// TwinCAT 3 PLC project MqttTest
// Title: MqttTest
// Company: FactoryAutomation
// Author: Filippo Boido
// ProjectVersion: 1.4.2.8
// ProgramVersion: 3.1.4023.0
// libraries:
//   ChainControllerLib, * (FactoryAutomation)
//   MqttFramework, * (FactoryAutomation)
//   StateMachineLib, * (FactoryAutomation)
//   StepWorkerLib, * (FactoryAutomation)
//   Tc2_Standard, * (Beckhoff Automation GmbH)
//   Tc2_System, * (Beckhoff Automation GmbH)
//   Tc3_Module, * (Beckhoff Automation GmbH)
//   VisuSymbols,3.5.10.0,System
// project tree:
//   / GlobalTextList.TcGTLO (not stored), PlcTask.TcTTO, Version.TcPOU, Visualisierungsmanager.TcVMO (not stored)
//   POUs/Basic/Conveyors/ BeltConveyor.TcPOU, Conveyor.TcPOU, PalletizerConveyor.TcPOU, RollerConveyor.TcPOU
//   POUs/Basic/Cylinder/ Cylinder.TcPOU
//   POUs/Basic/Elevator/ Elevator.TcPOU, PalletizerElevator.TcPOU
//   POUs/Basic/Sensor/ Sensor.TcPOU
//   POUs/HeavyModules/LineRegulator/ SM_LineRegulator.TcPOU
//   POUs/HeavyModules/TransferLine/ TL_BUSY.TcDUT, TL_RollerConveyors.TcDUT (not stored), SM_TransferLine.TcPOU
//   POUs/HeavyModules/TransferLine/StepChains/BeltConveyors/ SC_ACTUATOR_BeltConveyors.TcDUT (not stored), SC_BUSY_BeltConveyors.TcDUT, SC_SENSOR_BeltConveyors.TcDUT (not stored), SC_BeltConveyors.TcPOU
//   POUs/HeavyModules/TransferLine/StepChains/PostPalletizer/ SC_PostPalletizer.TcPOU
//   POUs/HeavyModules/TransferLine/StepChains/PrePalletizer/ SC_PrePalletizer.TcPOU
//   POUs/LightModules/PresenceDetector/ PresenceDetector.TcPOU
//   POUs/LightModules/Turntable/ Turntable.TcPOU
//   POUs/Main/ MAIN_BUSY.TcDUT (not stored), MAIN.TcPOU
//   POUs/MediumModules/Palletizer/ PAL_Busy.TcDUT, SM_Palletizer.TcPOU
//   POUs/MediumModules/Palletizer/StepChains/FirstFloor/ SC_BUSY_FirstFloor.TcDUT (not stored), SC_FirstFloor.TcPOU
//   POUs/MediumModules/Palletizer/StepChains/SecondFloor/ SC_BUSY_SecondFloor.TcDUT, SC_SecondFloor.TcPOU
//   POUs/ Visu.TcPOU (not stored)
//   VISUs/ Visualization.TcVIS
// real-time tasks:
//   TASK PlcTask: cycle T#10ms, priority 20, ADS port 350

CONFIGURATION MqttTest
    RESOURCE PLC ON TwinCAT3
        TASK PlcTask(INTERVAL := T#10ms, PRIORITY := 20);
        PROGRAM MAIN WITH PlcTask : MAIN;
    END_RESOURCE
END_CONFIGURATION

// ---- POUs/HeavyModules/TransferLine/TL_BUSY.TcDUT

TYPE TL_BUSY :
(
	eTlBusyStart := 0,
	eTlStartEntranceConveyor,
	eTlStartUpwardsConveyor,
	eTlExecutePalletizer,
	eTlSignalError
)UINT;
END_TYPE

// ---- POUs/HeavyModules/TransferLine/StepChains/BeltConveyors/SC_BUSY_BeltConveyors.TcDUT

TYPE SC_BUSY_BeltConveyors :
(
	eBusySCStart := 0,
	eStartEntranceConveyor,
	eStartUpwardsConveyor,
	eExecutePalletizer,
	eStopEntranceConveyor,
	eWaitForPalletizer,
	eSignalError
)UINT;
END_TYPE

// ---- POUs/MediumModules/Palletizer/PAL_Busy.TcDUT

TYPE PAL_Busy :
(
	ePALStart := 0
	
	
);
END_TYPE

// ---- POUs/MediumModules/Palletizer/StepChains/SecondFloor/SC_BUSY_SecondFloor.TcDUT

TYPE SC_BUSY_SecondFloor :
(
	eSecondFloorStart := 0,
	eActivateTurn,
	eActivateBeltForw,
	eWaitForPackages,
	ePushPackages,
	eRetractPusher,
	eClamp,
	eRetractClamper,
	eWaitForPallet,
	eOpenPlate,
	eClosePlate,
	eElevatorUp,
	eElevatorDown,
	eStartChains,
	eStopChains,
	eWaitForFirstFloor,
	eSyncWithFirstFloor,
	eSecondFloorDone
);
END_TYPE

// ---- POUs/Main/MAIN.TcPOU
PROGRAM MAIN
VAR
 aTransferLines  : ARRAY[1..3] OF SM_TransferLine;
 fbLineRegulator : SM_LineRegulator;
 fbSymbolPathStorage : SymbolPathStorage;
 fbMainStepWorker : FB_StepWorker;
END_VAR

aTransferLines[1]();
aTransferLines[2]();
aTransferLines[3]();
fbLineRegulator();

CASE fbMainStepWorker.uiStep OF
	
	eMainWaitStart:
	
		IF Visu.bStartTL1
		THEN
			aTransferLines[1].Execute();
		END_IF
		
		IF Visu.bStartTL2
		THEN
			aTransferLines[2].Execute();
		END_IF
		
		IF Visu.bStartTL3
		THEN
			aTransferLines[3].Execute();
		END_IF
		
		
	
END_CASE

END_PROGRAM

// ---- POUs/HeavyModules/TransferLine/SM_TransferLine.TcPOU
FUNCTION_BLOCK SM_TransferLine EXTENDS StateMachine
VAR_INPUT CONSTANT
	sTLMqttName : STRING;
END_VAR
VAR_OUTPUT
END_VAR
VAR
	
	aRollerConveyors : ARRAY[1..3] OF RollerConveyor;
	fbChainController : FB_ChainController;
	
	fbPalletizer : SM_Palletizer;
	fbStepWorkerReady : FB_StepWorker;
	fbStepWorkerBusy : FB_StepWorker;

	scBeltConveyors : 
		SC_BeltConveyors := 
		(
			sChainName  := 'scBeltConveyors',
			rChainController := fbChainController
		);
		
	scPostPalletizer : 
		SC_PostPalletizer := 
		(
			sChainName  := 'scPostPalletizer',
			rChainController := fbChainController
		);
		
	scPrePalletizer : 
		SC_PrePalletizer := 
		(
			sChainName  := 'scPrePalletizer',
			rChainController := fbChainController
		);
 
	uiPackageCounter : UINT;
	i : UINT;
	bPackageOnTheWay : BOOL;
	
END_VAR

SUPER^();
fbPalletizer(ioChainController := fbChainController);
scBeltConveyors(bAllPartsPresent := fbPalletizer.bAllPartsPresent);
scPrePalletizer();
scPrePalletizer.bPalletizerRequest := fbPalletizer.scFirstFloor.bPalletizerRequest;
fbPalletizer.scFirstFloor.bIncomingPallet := scPrePalletizer.bSentToPalletizer;
scPostPalletizer();

METHOD PROTECTED Busy : BOOL
VAR_INPUT
END_VAR
CASE fbStepWorkerBusy.uiStep OF
	eTlStartUnits:
		scBeltConveyors.bExecute := TRUE;
		scPrePalletizer.bExecute := TRUE;
		scPostPalletizer.bExecute := TRUE;
		fbPalletizer.bExecute := TRUE;
		fbStepWorkerBusy.mNextStep(eTlCheckUnits);
	eTlCheckUnits:
		IF scBeltConveyors.eStateMachine = E_StateMachine.eError
		THEN
			fbStepWorkerBusy.mNextStep(eTlSignalError);
		END_IF
	eTlSignalError:
		Fault();
END_CASE
END_METHOD

METHOD PROTECTED  Error : BOOL
VAR_INPUT
END_VAR
END_METHOD

METHOD PROTECTED  Idle : BOOL
VAR_INPUT
END_VAR
Start();
END_METHOD

METHOD PROTECTED  Init : BOOL
VAR_INPUT
END_VAR
fbChainController
	.addChain(itfChain := scBeltConveyors)
	.addChain(itfChain := scPostPalletizer)
	.addChain(itfChain := scPrePalletizer);
	
	
Start();
END_METHOD

METHOD PROTECTED  Prepare : BOOL
VAR_INPUT
END_VAR
END_METHOD

METHOD PROTECTED  Ready : BOOL
VAR_INPUT
END_VAR
END_METHOD

METHOD PROTECTED  Waiting : BOOL
VAR_INPUT
END_VAR
END_METHOD

END_FUNCTION_BLOCK

// ---- POUs/Basic/Conveyors/RollerConveyor.TcPOU
FUNCTION_BLOCK RollerConveyor EXTENDS Conveyor
VAR_INPUT
END_VAR
VAR_OUTPUT
END_VAR
VAR
END_VAR

Super^();

END_FUNCTION_BLOCK

// ---- POUs/Basic/Conveyors/Conveyor.TcPOU
FUNCTION_BLOCK Conveyor 
VAR_INPUT
END_VAR

VAR_OUTPUT
	bStart  : BOOL;
END_VAR
VAR
	fbStart : BoolOut;
END_VAR

bStart := fbStart.getValue;

PROPERTY getStart : I_StepCondition
GET
getStart := fbStart;
END_GET
END_PROPERTY

METHOD Off : BOOL
VAR_INPUT
END_VAR
fbStart.setValue := FALSE;
END_METHOD

METHOD On : BOOL
VAR_INPUT
END_VAR
fbStart.setValue := TRUE;
END_METHOD

END_FUNCTION_BLOCK

// ---- POUs/MediumModules/Palletizer/SM_Palletizer.TcPOU
FUNCTION_BLOCK SM_Palletizer EXTENDS StateMachine
VAR_IN_OUT
	ioChainController : FB_ChainController;
END_VAR
VAR_OUTPUT
	
	bAllPartsPresent: BOOL;	
	
END_VAR
VAR

	fbDoneCycle : BoolOut;
	fbStepWorkerBusy : FB_StepWorker;
	
	scFirstFloor : SC_FirstFloor :=
	(
		sChainName := 'scFirstFloor',
		rChainController := ioChainController
	);
	
	scSecondFloor : SC_SecondFloor :=
	(
		sChainName := 'scSecondFloor',
		rChainController := ioChainController
	);
END_VAR

SUPER^();
scFirstFloor();
scSecondFloor();

bAllPartsPresent := scSecondFloor.bAllPartsPresent;
scSecondFloor.bPlateOpen := scFirstFloor.bPlateOpen;

METHOD PROTECTED   Busy : BOOL
VAR_INPUT
END_VAR
scFirstFloor(bExecute := TRUE);
scSecondFloor(bExecute := TRUE);
END_METHOD

METHOD PROTECTED  Error : BOOL
VAR_INPUT
END_VAR
END_METHOD

PROPERTY getDoneCycle : I_StepCondition
GET
getDoneCycle := fbDoneCycle;
END_GET
END_PROPERTY

METHOD PROTECTED  Idle : BOOL
VAR_INPUT
END_VAR
END_METHOD

METHOD PROTECTED  Init : BOOL
VAR_INPUT
END_VAR
ioChainController
	.addChain(itfChain := scFirstFloor)
	.addChain(itfChain := scSecondFloor);
	
Start();
END_METHOD

METHOD PROTECTED  Prepare : BOOL
VAR_INPUT
END_VAR
END_METHOD

METHOD PROTECTED  Ready : BOOL
VAR_INPUT
END_VAR
END_METHOD

METHOD PROTECTED  Waiting : BOOL
VAR_INPUT
END_VAR
END_METHOD

END_FUNCTION_BLOCK

// ---- POUs/MediumModules/Palletizer/StepChains/FirstFloor/SC_FirstFloor.TcPOU
FUNCTION_BLOCK SC_FirstFloor EXTENDS FB_Chain
VAR_INPUT
	bExecute : BOOL;
	bIncomingPallet : BOOL;
	bPostPalletizerRequestGranted : BOOL;
END_VAR
VAR_OUTPUT
	bPlateOpen : BOOL;
	bPalletizerRequest : BOOL;
	bSentToPostPalletizer : BOOL;
	bPostPalletizerDeliveryRequest : BOOL;
END_VAR
VAR
	fbPallChainConveyor : PalletizerConveyor;
	fbPallElevator : PalletizerElevator;
	fbPlateCyl : Cylinder;
	fbPlateLimitSen : Sensor;
	fbElevatorFrontLimit : Sensor;
	fbElevatorBackLimit : Sensor;
END_VAR

SUPER^();
bPlateOpen := fbPlateCyl.bExtended;
fbPallChainConveyor();
fbPallElevator();
fbPlateCyl();
fbPlateLimitSen();

METHOD PROTECTED   Busy : BOOL
VAR_INPUT
END_VAR

		
fbStepWorkerBusy();
CASE fbStepWorkerBusy.uiStep OF
	
	0: 
		fbPallChainConveyor.On();
		fbStepWorkerBusy
			.mAddCondition(itfStepCondition := fbElevatorBackLimit.getSignal)
			.mAddCondition(itfStepCOndition := fbElevatorFrontLimit.getSignal)
			.mNextStep(10);
			
	10: 
	
		fbPallChainConveyor.Off();
		bPalletizerRequest := FALSE;
		IF rChainController
			.releaseCheck(THIS^)
			.releaseFromChain(sChainReleasing := 'scSecondFloor', THIS^)
			.releaseResult(THIS^) 
		THEN
			fbStepWorkerBusy.mNextStep(20);
		END_IF

	20:
	
		fbPallElevator.MoveUp();
		fbStepWorkerBusy
			.mSetTimer(T#1S)
			.mNextStep(30);
			
	30:
	
		IF NOT fbPallElevator.isMoving
		THEN
			fbStepWorkerBusy.mNextStep(40);
		END_IF
		
	40:
	
		fbPlateCyl.Extend();
		fbStepWorkerBusy
			.mSetTimer(T#1S)
			.mNextStep(50);
			
	50:
	
		//Plate is open
		IF fbPlateLimitSen.bSignal
		THEN
			fbStepWorkerBusy
				.mSetTimer(T#1S)
				.mNextStep(60);
		END_IF
		
	60:
		fbPlateCyl.Retract();
		fbStepWorkerBusy
			.mSetTimer(T#1S)
			.mNextStep(70);
			
	70:
	
		//Plate is closed
		IF fbPlateLimitSen.bSignal
		THEN
			fbStepWorkerBusy.mNextStep(80);
		END_IF
		
	80:
	
		rChainController.releaseForChain('scSecondFloor', THIS^);	
		fbPallElevator.MoveDown();
		fbStepWorkerBusy.mNextStep(90);
		
	90:

		IF NOT fbPallElevator.isMoving
		THEN
			rChainController.releaseForChain('scPostPalletizer', THIS^);
			fbStepWorkerBusy.mNextStep(100);
		END_IF	
		
	100:
	
		IF rChainController
			.releaseCheck(THIS^)
			.releaseFromChain(sChainReleasing := 'scPostPalletizer', THIS^)
			.releaseResult(THIS^) 
		THEN

			fbPallChainConveyor.On();
			fbStepWorkerReady.mNextStep(110);
		END_IF
		
	110:
	
		
		
		IF NOT fbElevatorBackLimit.bSignal
			AND NOT fbElevatorFrontLimit.bSignal
		THEN
		
			Done();
			fbStepWorkerReady.mNextStep(0);
		END_IF

END_CASE
END_METHOD

METHOD PROTECTED  Error : BOOL
VAR_INPUT
END_VAR
END_METHOD

METHOD PROTECTED  Idle : BOOL
VAR_INPUT
END_VAR
END_METHOD

METHOD PROTECTED  Init : BOOL
VAR_INPUT
END_VAR
Start();
END_METHOD

METHOD PROTECTED  Prepare : BOOL
VAR_INPUT
END_VAR
END_METHOD

METHOD PROTECTED  Ready : BOOL
VAR_INPUT
END_VAR

fbStepWorkerReady();
CASE fbStepWorkerReady.uiStep OF
	
	0: 
	
		IF bExecute THEN
			fbStepWorkerReady.mNextStep(10);
		END_IF
		
	10:

		IF NOT fbElevatorFrontLimit.bSignal
			AND NOT fbElevatorBackLimit.bSignal 
		THEN
			bPalletizerRequest := TRUE;
			fbStepWorkerReady.mNextStep(20);
		END_IF
		
	20:
	
		IF bIncomingPallet
		THEN
			fbStepWorkerReady.mNextStep(0);
			Execute();
		END_IF
		
		
END_CASE
END_METHOD

METHOD PROTECTED  Waiting : BOOL
VAR_INPUT
END_VAR
END_METHOD

END_FUNCTION_BLOCK

// ---- POUs/Basic/Conveyors/PalletizerConveyor.TcPOU
FUNCTION_BLOCK PalletizerConveyor EXTENDS Conveyor
VAR_INPUT
END_VAR
VAR_OUTPUT
	bStartBackward : BOOL;
END_VAR
VAR	
	fbStartBackward : BoolOut;
END_VAR

SUPER^();
bStartBackward := fbStartBackward.getValue;

PROPERTY getStartBackward : BoolOut
GET
getStartBackward := fbStartBackward;
END_GET
END_PROPERTY

END_FUNCTION_BLOCK

// ---- POUs/Basic/Elevator/PalletizerElevator.TcPOU
FUNCTION_BLOCK PalletizerElevator EXTENDS Elevator
VAR_INPUT
END_VAR
VAR_OUTPUT
	isMoving : BOOL;
END_VAR
VAR
	fbElevatorMoving : Sensor;
	
END_VAR

isMoving := fbElevatorMoving.bSignal;

METHOD MoveDown : BOOL
VAR_INPUT
END_VAR
END_METHOD

METHOD MoveUp : BOOL
VAR_INPUT
END_VAR
END_METHOD

METHOD StepDown : BOOL
VAR_INPUT
END_VAR
END_METHOD

METHOD StepUp : BOOL
VAR_INPUT
END_VAR
END_METHOD

END_FUNCTION_BLOCK

// ---- POUs/Basic/Elevator/Elevator.TcPOU
FUNCTION_BLOCK Elevator
VAR_INPUT
END_VAR
VAR_OUTPUT
END_VAR
VAR
END_VAR

END_FUNCTION_BLOCK

// ---- POUs/Basic/Sensor/Sensor.TcPOU
FUNCTION_BLOCK Sensor
VAR_INPUT
END_VAR
VAR_OUTPUT
	bSignal  : BOOL;
END_VAR
VAR
	fbSignal : BoolIn;
END_VAR

bSignal := fbSignal.getValue;

PROPERTY getSignal : BoolIn
GET
getSignal := fbSignal;
END_GET
END_PROPERTY

END_FUNCTION_BLOCK

// ---- POUs/Basic/Cylinder/Cylinder.TcPOU
FUNCTION_BLOCK Cylinder 
VAR_INPUT
END_VAR
VAR_OUTPUT
	bExtended : BOOL;
	bExtend : BOOL;
END_VAR
VAR
	fbExtendedSignal : BoolIn;
	fbExtend : BoolOut;
END_VAR

bExtended := fbExtendedSignal.getValue;
bExtend := fbExtend.getValue;

PROPERTY getExtend : BoolOut
GET
getExtend := fbExtend;
END_GET
END_PROPERTY

END_FUNCTION_BLOCK

// ---- POUs/MediumModules/Palletizer/StepChains/SecondFloor/SC_SecondFloor.TcPOU
FUNCTION_BLOCK SC_SecondFloor EXTENDS FB_Chain
VAR_INPUT
	bExecute : BOOL;
	bPlateOpen : BOOL;
END_VAR
VAR_OUTPUT
	bAllPartsPresent: BOOL;	
END_VAR
VAR
	fbPallBeltConveyor : PalletizerConveyor;
	fbPushCyl : Cylinder;
	fbTurnCyl : Cylinder;
	
	fbClampCyl : Cylinder;
	fbClampedSen : Sensor;
	
	fbPusherLimitSen : Sensor;
	fbPresenceDetector : PresenceDetector;
	iCycle : INT;
END_VAR

SUPER^();

fbPushCyl();
fbTurnCyl();

fbClampCyl();
fbPallBeltConveyor();
fbPresenceDetector(bAllPartsPresent => bAllPartsPresent);

METHOD PROTECTED   Busy : BOOL
VAR_INPUT
END_VAR
fbStepWorkerBusy();
CASE fbStepWorkerBusy.uiStep OF
	
	eSecondFloorStart: //send release to scBeltConveyor
	
		iCycle := iCycle + 1;
		rChainController.releaseForChain('scBeltConveyor', THIS^);
		fbStepWorkerBusy.mNextStep(10);
		
	10: //wait for release from scBeltConveyor to start actuators
	
		IF rChainController
			.releaseCheck(THIS^)
			.releaseFromChain(sChainReleasing := 'scBeltConveyor', THIS^)
			.releaseResult(THIS^) 
		THEN
			fbStepWorkerBusy.mNextStep(20);
		END_IF
	
		
	20: //wait for packages
		
		fbTurnCyl.Extend();
		fbPallBeltConveyor.On();
		IF fbPresenceDetector.bAllPartsPresent
		THEN
			bAllPartsPresent := TRUE;
			fbPallBeltConveyor.Off();
			fbStepWorkerBusy.mNextStep(ePushPackages);
		END_IF	
		
	ePushPackages:
	
		fbPushCyl.Extend();
		
		fbStepWorkerBusy
			.mSetTimer(T#2S)
			.mNextStep(eRetractPusher);
		
	eRetractPusher:
	
		fbPushCyl.Retract();
		
		fbStepWorkerBusy
			.mSetTimer(T#2S)
			.mNextStep(eClamp);
			
	eClamp:
	
		fbClampCyl.Extend();
		fbStepWorkerBusy
			.mSetTimer(T#2S)
			.mNextStep(eRetractClamper);
			
	eRetractClamper:
	
		
		fbClampCyl.Retract();
		IF iCycle = 1
		THEN
			fbStepWorkerBusy
				.mSetTimer(T#2S)
				.mNextStep(eSecondFloorDone);
		ELSE
			iCycle := 0;
			fbStepWorkerBusy.mNextStep(eSyncWithFirstFloor);
		END_IF
		
	eSyncWithFirstFloor:
	
		rChainController.releaseForChain('scFirstFloor', THIS^);	
		fbStepWorkerBusy.mNextStep(eWaitForFirstFloor);
	
	eWaitForFirstFloor:
	
		IF rChainController
			.releaseCheck(THIS^)
			.releaseFromChain(sChainReleasing := 'scFirstFloor', THIS^)
			.releaseResult(THIS^) 
		THEN
			fbStepWorkerBusy.mNextStep(eSecondFloorDone);
		END_IF
		
	eSecondFloorDone:
		fbStepWorkerBusy.mNextStep(eSecondFloorStart);
		Done();	
	
END_CASE
END_METHOD

METHOD PROTECTED  Error : BOOL
VAR_INPUT
END_VAR
END_METHOD

METHOD PROTECTED  Idle : BOOL
VAR_INPUT
END_VAR
END_METHOD

METHOD PROTECTED  Init : BOOL
VAR_INPUT
END_VAR
Start();
END_METHOD

METHOD PROTECTED  Prepare : BOOL
VAR_INPUT
END_VAR
END_METHOD

METHOD PROTECTED  Ready : BOOL
VAR_INPUT
END_VAR

fbStepWorkerReady();
CASE fbStepWorkerReady.uiStep OF
	
	0: 
	
		IF bExecute THEN
			fbStepWorkerReady.mNextStep(10);
		END_IF
		
	10:
		
		IF NOT fbPresenceDetector.bAllPartsPresent
			AND NOT bPlateOpen
		THEN
			rChainController.releaseForChain('scBeltConveyor', THIS^);	
			fbStepWorkerReady.mNextStep(20);	
		END_IF
	
	20:
		
		IF rChainController
			.releaseCheck(THIS^)
			.releaseFromChain(sChainReleasing := 'scBeltConveyor', THIS^)
			.releaseResult(THIS^) 
		THEN
			fbStepWorkerBusy.mNextStep(0);
			Execute();
		END_IF
		
END_CASE
END_METHOD

METHOD PROTECTED  Waiting : BOOL
VAR_INPUT
END_VAR
END_METHOD

END_FUNCTION_BLOCK

// ---- POUs/LightModules/PresenceDetector/PresenceDetector.TcPOU
FUNCTION_BLOCK PresenceDetector
VAR_INPUT
END_VAR
VAR_OUTPUT
	bAllPartsPresent : BOOL;
END_VAR
VAR
	aSensors : ARRAY[1..3] OF Sensor;
	fbTimer : TON;
	i: INT;
END_VAR

aSensors[1]();
aSensors[2]();
aSensors[3]();
fbTimer(
	IN:= aSensors[1].bSignal
		AND aSensors[2].bSignal
		AND aSensors[3].bSignal,
	PT:=T#2S
);
IF fbTimer.Q
THEN
	bAllPartsPresent := TRUE;
ELSE
	bAllPartsPresent :=FALSE;
END_IF

END_FUNCTION_BLOCK

// ---- POUs/HeavyModules/TransferLine/StepChains/BeltConveyors/SC_BeltConveyors.TcPOU
FUNCTION_BLOCK SC_BeltConveyors EXTENDS FB_Chain
VAR_INPUT
	bExecute : BOOL;
	bAllPartsPresent : BOOL;
END_VAR
VAR_OUTPUT
END_VAR
VAR
	aBeltConveyors : ARRAY[1..2] OF BeltConveyor;
	fbCounterSensor : Sensor;
	i : INT;
	uiPackageCounter : UINT;
	fbTrig : R_TRIG;
	
END_VAR

SUPER^();
fbCounterSensor();
fbTrig(CLK := fbCounterSensor.bSignal);
IF fbTrig.Q
THEN
	uiPackageCounter := uiPackageCounter + 1;
END_IF
FOR i := 1 TO (eMaxNumBeltConveyors - 1)
DO
	
	aBeltConveyors[i]();

END_FOR

METHOD PROTECTED Busy : BOOL
VAR_INPUT
END_VAR
VAR
	iStepCondition : I_StepCondition;
END_VAR
fbStepWorkerBusy();

CASE fbStepWorkerBusy.uiStep OF

	eBusySCStart: 
		THIS^.aBeltConveyors[eBeltConveyorEntrance].On();
		
		fbStepWorkerBusy.mNextStep(10);
		
	10:
		//As Soon as the first package reaches the counter sensor
		//the second floor of the palletizer is informed
		//consequently the second floor of the palletizer will go in busy mode.
		IF uiPackageCounter = 1
		THEN
			THIS^.aBeltConveyors[eBeltConveyorUpwards].On();
			
			fbStepWorkerBusy.mNextStep(15);
		END_IF
		
	15:
		IF uiPackageCounter = 3
		THEN
			uiPackageCounter := 0;
			fbStepWorkerBusy.mNextStep(20);
		END_IF
	20:
		fbStepWorkerBusy
				.mSetTimer(T#1s)
				.mNextStep(30);
	30:
		THIS^.aBeltConveyors[eBeltConveyorEntrance].Off();
		IF bAllPartsPresent
		THEN
			THIS^.aBeltConveyors[eBeltConveyorUpwards].Off();
			Done();
			fbStepWorkerBusy.mNextStep(0);
		END_IF
		
	40:
	
		
		(*
		//At start we check how many packages have passed the fbCounterSensor
		IF uiPackageCounter < 3
		THEN
		
			//activate the conveyors
			fbStepWorkerBusy.mNextStep(eStartEntranceConveyor);
			
		ELSIF uiPackageCounter = 3
		 AND NOT ioPalletizer.bAllPartsPresent
		 AND aBeltConveyors[eBeltConveyorEntrance].bStart
		THEN
 			//A package needs to reach the palletizer or a sensor is malfunctioning		
			fbStepWorkerBusy
				.mSetTimer(T#1s)
				.mNextStep(eStopEntranceConveyor);
				
		ELSIF uiPackageCounter = 3
		 AND ioPalletizer.bAllPartsPresent
	 	THEN
			//Execute the Palletizer
			uiPackageCounter := 0;
			aBeltConveyors[eBeltConveyorUpwards].Off();
			fbStepWorkerBusy.mNextStep(eWaitForPalletizer);
		ELSIF uiPackageCounter > 3
		THEN
			//Error
		END_IF
		
	eStartEntranceConveyor:
		
		aBeltConveyors[eBeltConveyorEntrance].On();
		fbStepWorkerBusy.mAddCondition(fbCounterSensor.getSignal);
		fbStepWorkerBusy.mNextStep(eStartUpwardsConveyor);

	eStartUpwardsConveyor:
	
		
		aBeltConveyors[eBeltConveyorUpwards].On();
		fbStepWorkerBusy.mNextStep(eExecutePalletizer);
			 
	eExecutePalletizer:
		 
		ioPalletizer.Execute();	
		fbStepWorkerBusy.mNextStep(eBusySCStart);
	
	eStopEntranceConveyor:
		aBeltConveyors[eBeltConveyorEntrance].Off();
		fbStepWorkerBusy.mNextStep(eExecutePalletizer);
		
	eWaitForPalletizer:
	
		 fbStepWorkerBusy.mAddCondition(ioPalletizer.getDoneCycle);
		 fbStepWorkerBusy.mNextStep(eBusySCStart);
		 
	eSignalError:
	
		fbStepWorkerBusy.mNextStep(eBusySCStart);
		Fault();	
		*)	
END_CASE
END_METHOD

METHOD PROTECTED  Error : BOOL
VAR_INPUT
END_VAR
VAR
	i : INT;
END_VAR
FOR i := 1 TO 3 
DO

	aBeltConveyors[i].Off();
	
END_FOR
END_METHOD

METHOD PROTECTED  Idle : BOOL
VAR_INPUT
END_VAR
END_METHOD

METHOD PROTECTED  Init : BOOL
VAR_INPUT
END_VAR
Start();
END_METHOD

METHOD PROTECTED  Prepare : BOOL
VAR_INPUT
END_VAR
END_METHOD

METHOD PROTECTED  Ready : BOOL
VAR_INPUT
END_VAR
fbStepWorkerReady();
CASE fbStepWorkerReady.uiStep OF
	
	0: 
	
		IF bExecute THEN
			fbStepWorkerReady.mNextStep(10);
		END_IF
		
	10:
	
		IF rChainController
			.releaseCheck(THIS^)
			.releaseFromChain(sChainReleasing := 'scSecondFloor', THIS^)
			.releaseResult(THIS^) 
		THEN
			Execute();
			rChainController.releaseForChain('scSecondFloor', THIS^);		
			fbStepWorkerReady.mNextStep(0);
		END_IF
	
		
	
END_CASE
END_METHOD

METHOD PROTECTED  Waiting : BOOL
VAR_INPUT
END_VAR
END_METHOD

END_FUNCTION_BLOCK

// ---- POUs/Basic/Conveyors/BeltConveyor.TcPOU
FUNCTION_BLOCK BeltConveyor EXTENDS Conveyor
VAR_INPUT
END_VAR
VAR_OUTPUT
END_VAR
VAR
END_VAR

Super^();

END_FUNCTION_BLOCK

// ---- POUs/HeavyModules/TransferLine/StepChains/PostPalletizer/SC_PostPalletizer.TcPOU
FUNCTION_BLOCK SC_PostPalletizer EXTENDS FB_Chain
VAR_INPUT
	bExecute : BOOL;
	bPalletizerDeliveryRequest : BOOL;
	sTLMqttName : STRING;
END_VAR
VAR_OUTPUT
	bGrantDeliveryPermission : BOOL;
END_VAR
VAR
	
	fbPalletAvailable : Sensor;
	fbRollConveyor : RollerConveyor;
	
END_VAR

SUPER^();
fbPalletAvailable();
fbRollConveyor();

METHOD PROTECTED   Busy : BOOL
VAR_INPUT
END_VAR
VAR
	stMqttPayload : ST_MqttPayload;
	messageIndex : UINT;
END_VAR
fbStepWorkerBusy();
CASE fbStepWorkerBusy.uiStep OF
	
	0: 
		THIS^.fbRollConveyor.On();
		rChainController.releaseForChain('scFirstFloor', THIS^);
		fbStepWorkerBusy.mNextStep(10);
		
	10:
		IF THIS^.fbPalletAvailable.bSignal
		THEN
			THIS^.fbRollConveyor.Off();
			fbStepWorkerBusy.mNextStep(20);
		END_IF
	
	20: 
		
		//Mqtt exchange
		IF Ads.fbMqttClient.Publish(sTLMqttName,stMqttPayload)
		THEN
			fbStepWorkerBusy.mNextStep(30);
		END_IF
	
	30:
	
		messageIndex := ADS.fbMqttClient.isNewMessage(sTLMqttName);
		IF messageIndex > 0
		THEN
			stMqttPayload := Ads.fbMqttClient.getNewMessage(messageIndex);
			fbStepWorkerBusy.mNextStep(40);
		END_IF
		
	40:
	
		THIS^.fbRollConveyor.On();
		fbStepWorkerBusy
			.mSetTimer(T#2S)
			.mNextStep(50);
			
	50:
		
		THIS^.fbRollConveyor.Off();
		Done();
		fbStepWorkerBusy.mNextStep(0);
		
END_CASE
END_METHOD

METHOD PROTECTED  Error : BOOL
VAR_INPUT
END_VAR
END_METHOD

METHOD PROTECTED  Idle : BOOL
VAR_INPUT
END_VAR
END_METHOD

METHOD PROTECTED  Init : BOOL
VAR_INPUT
END_VAR
IF ADS.fbMqttClient.Subscribe(sTopic := sTLMqttName)
THEN			
	Start();
END_IF
END_METHOD

METHOD PROTECTED  Prepare : BOOL
VAR_INPUT
END_VAR
END_METHOD

METHOD PROTECTED  Ready : BOOL
VAR_INPUT
END_VAR

fbStepWorkerReady();
CASE fbStepWorkerReady.uiStep OF
	
0:

	IF bExecute
		AND NOT fbPalletAvailable.bSignal
	THEN
		fbStepWorkerReady.mNextStep(10);
	END_IF
		
10:
	IF rChainController
		.releaseCheck(THIS^)
		.releaseFromChain(sChainReleasing := 'scFirstFloor', THIS^)
		.releaseResult(THIS^) 
	THEN
		fbStepWorkerReady.mNextStep(0);
		Execute();
	END_IF
	
END_CASE
END_METHOD

METHOD PROTECTED  Waiting : BOOL
VAR_INPUT
END_VAR
END_METHOD

END_FUNCTION_BLOCK

// ---- POUs/HeavyModules/TransferLine/StepChains/PrePalletizer/SC_PrePalletizer.TcPOU
FUNCTION_BLOCK SC_PrePalletizer EXTENDS FB_Chain
VAR_INPUT
	bPalletizerRequest : BOOL;
	bExecute : BOOL;
END_VAR
VAR_OUTPUT
	bSentToPalletizer : BOOL;
	bPalletAvailable : BOOL;
END_VAR
VAR
	fbRollConvEntrance : RollerConveyor;
	fbRollConvPrePallet : RollerConveyor;
	fbPalletAvailable : Sensor;
END_VAR

SUPER^();
fbPalletAvailable();
bPalletAvailable := fbPalletAvailable.bSignal;

METHOD PROTECTED   Busy : BOOL
VAR_INPUT
END_VAR
fbStepWorkerBusy();
CASE fbStepWorkerBusy.uiStep OF
	
	0: 
		fbRollConvEntrance.On();
		fbRollConvPrePallet.On();
		IF NOT bPalletAvailable
		THEN
			bSentToPalletizer := TRUE;
			fbStepWorkerBusy.mNextStep(10);
		END_IF

	10:
		IF NOT bPalletizerRequest
		THEN
		
			bSentToPalletizer := FALSE;
			fbRollConvPrePallet.Off();
			fbStepWorkerBusy.mNextStep(0);
			
			Done();
			
		ELSIF bPalletAvailable
		THEN
			fbRollConvEntrance.Off();
		END_IF
		
END_CASE
END_METHOD

METHOD PROTECTED  Error : BOOL
VAR_INPUT
END_VAR
END_METHOD

METHOD PROTECTED  Idle : BOOL
VAR_INPUT
END_VAR
END_METHOD

METHOD PROTECTED  Init : BOOL
VAR_INPUT
END_VAR
Start();
END_METHOD

METHOD PROTECTED  Prepare : BOOL
VAR_INPUT
END_VAR
END_METHOD

METHOD PROTECTED  Ready : BOOL
VAR_INPUT
END_VAR

fbStepWorkerReady();
CASE fbStepWorkerReady.uiStep OF
	
	0:
		IF bExecute
		THEN
			fbStepWorkerReady.mNextStep(5);
		END_IF
		
	5: 
		IF NOT bPalletAvailable
		THEN
			fbRollConvEntrance.On();
		ELSIF bPalletAvailable
		THEN
			fbRollConvEntrance.Off();
			fbStepWorkerReady.mNextStep(10);
		END_IF
		
	10:
		IF bPalletizerRequest
		THEN
			fbStepWorkerReady.mNextStep(0);
			Execute();
		END_IF
		
END_CASE
END_METHOD

METHOD PROTECTED  Waiting : BOOL
VAR_INPUT
END_VAR
END_METHOD

END_FUNCTION_BLOCK

// ---- POUs/HeavyModules/LineRegulator/SM_LineRegulator.TcPOU
FUNCTION_BLOCK SM_LineRegulator EXTENDS StateMachine
VAR_INPUT
END_VAR
VAR_OUTPUT
END_VAR
VAR
	fbTurntable : Turntable;

	aRollerConveyors : ARRAY[1..3] OF RollerConveyor;
	fbReadyStepWorker : FB_StepWorker;
	fbBusyStepWorker : FB_StepWorker;
	fbInitStepWorker : FB_StepWorker;
	
	messageIndex : UINT;
	stMqttPayload : ST_MqttPayload;
	aSubscriptions : ARRAY[1..3] OF STRING;
	uiSubscriptionsCycler : UINT := 1;
END_VAR

SUPER^();
fbTurntable();
aRollerConveyors[1]();
aRollerConveyors[3]();

METHOD PROTECTED   Busy : BOOL
VAR_INPUT
END_VAR
fbBusyStepWorker();
CASE fbBusyStepWorker.uiStep OF

	0:
		aRollerConveyors[uiSubscriptionsCycler].On();
		CASE uiSubscriptionsCycler OF
		
			1:
				fbTurntable.RollPlus();
				fbTurntable.Turn();
			
			2:
				fbTurntable.RollPlus();
			
			3:
				fbTurntable.RollMinus();
				fbTurntable.Turn();
		END_CASE
		
		fbBusyStepWorker
			.mAddCondition(itfStepCondition := fbTurntable.fbBackLimit.getSignal)
			.mAddCondition(itfStepCondition := fbTurntable.fbFrontLimit.getSignal)
			.mNextStep(10);
	10:
	
		aRollerConveyors[uiSubscriptionsCycler].Off();
		CASE uiSubscriptionsCycler OF
		
			1:
				fbTurntable.StopRolling();			
				fbTurntable.UnTurn();
				fbBusyStepWorker
					.mSetTimer(T#2S)
					.mNextStep(20);
			
			2:
				fbBusyStepWorker.mNextStep(30);
			
			3:
				fbTurntable.StopRolling();
				fbTurntable.UnTurn();
				fbBusyStepWorker
					.mSetTimer(T#2S)
					.mNextStep(20);
		END_CASE
		
	20:
		fbTurntable.RollPlus();
		fbBusyStepWorker
			.mSetTimer(T#2S)
			.mNextStep(30);
	30:	
	
		IF NOT fbTurntable.fbBackLimit.bSignal
			AND NOT fbTurntable.fbFrontLimit.bSignal
		THEN
			fbBusyStepWorker
				.mSetTimer(T#2S)
				.mNextStep(40);
		END_IF
		
	40:
	
		fbBusyStepWorker.mNextStep(0);
		Done();
		
	
END_CASE
END_METHOD

METHOD PROTECTED  Error : BOOL
VAR_INPUT
END_VAR
END_METHOD

METHOD PROTECTED  Idle : BOOL
VAR_INPUT
END_VAR
END_METHOD

METHOD PROTECTED  Init : BOOL
VAR_INPUT
END_VAR
fbInitStepWorker();
CASE fbInitStepWorker.uiStep OF

	0: 
		IF ADS.fbAdsConnector.isConnected
		THEN
			fbInitStepWorker.mNextStep(10);
		END_IF
	10:
	
		IF ADS.fbMqttClient.Subscribe('TL1_Synch')
		THEN			
			fbInitStepWorker.mNextStep(20);
		END_IF
		
	20:
	
		IF ADS.fbMqttClient.Subscribe('TL2_Synch')
		THEN			
			fbInitStepWorker.mNextStep(30);
		END_IF
		
	30:
		
		IF ADS.fbMqttClient.Subscribe('TL3_Synch')
		THEN			
			Start();
		END_IF		
		
END_CASE
END_METHOD

METHOD PROTECTED  Prepare : BOOL
VAR_INPUT
END_VAR
END_METHOD

METHOD PROTECTED  Ready : BOOL
VAR_INPUT
END_VAR
VAR
	
END_VAR
fbReadyStepWorker();

IF uiSubscriptionsCycler = 3
THEN
	uiSubscriptionsCycler := 1;
ELSE
	uiSubscriptionsCycler := uiSubscriptionsCycler + 1;
END_IF

CASE fbReadyStepWorker.uiStep OF

	0: 
		IF NOT fbTurntable.bBackLimit
			AND NOT fbTurntable.bFrontLimit
		THEN
			fbReadyStepWorker.mNextStep(10);
		END_IF
		
	10:
	
		messageIndex := ADS.fbMqttClient.isNewMessage(aSubscriptions[uiSubscriptionsCycler]);
		IF messageIndex > 0
		THEN
			stMqttPayload := Ads.fbMqttClient.getNewMessage(messageIndex);
			fbReadyStepWorker.mNextStep(20);
		END_IF
		
	20:	
		Ads.fbMqttClient.Publish(aSubscriptions[uiSubscriptionsCycler],stMqttPayload);
		fbReadyStepWorker.mNextStep(0);
		Execute();
		
END_CASE
END_METHOD

METHOD PROTECTED  Waiting : BOOL
VAR_INPUT
END_VAR
END_METHOD

END_FUNCTION_BLOCK

// ---- POUs/LightModules/Turntable/Turntable.TcPOU
FUNCTION_BLOCK Turntable
VAR_INPUT



END_VAR
VAR_OUTPUT

	bTurn 		: BOOL;
	bRollPlus	: BOOL;
	bRollMinus 	: BOOL;
	bFrontLimit : BOOL;
	bBackLimit	: BOOL;
	
END_VAR
VAR

	fbFrontLimit : BoolIn;
	fbBackLimit : BoolIn;
	
	fbTurn : BoolOut;
	fbRollPlus : BoolOut;
	fbRollMinus : BoolOut;
	
END_VAR

bTurn := fbTurn.getValue;
bRollPlus := fbRollPlus.getValue;
bRollMinus := fbRollMinus.getValue;
bFrontLimit := fbFrontLimit.getValue;
bBackLimit	:= fbBackLimit.getValue;

METHOD RollMinus : BOOL
VAR_INPUT
END_VAR
fbRollMinus.setValue := TRUE;
fbRollPlus.setValue := FALSE;
END_METHOD

METHOD RollPlus : BOOL
VAR_INPUT
END_VAR
fbRollPlus.setValue := TRUE;
fbRollMinus.setValue := FALSE;
END_METHOD

METHOD StopRolling : BOOL
VAR_INPUT
END_VAR
fbRollMinus.setValue := FALSE;
fbRollPlus.setValue := FALSE;
END_METHOD

METHOD Turn : BOOL
VAR_INPUT
END_VAR
fbTurn.setValue := TRUE;
END_METHOD

METHOD Unturn : BOOL
VAR_INPUT
END_VAR
fbTurn.setValue := FALSE;
END_METHOD

END_FUNCTION_BLOCK

// ---- Version.TcPOU
PROGRAM Version
VAR
END_VAR

(*
1.0.1.1:	Boido	010120

Changed naming convention for main modules.
The first 2 letters give a hint on the inheritance relationship of the FB.

1.0.2.2:	Boido	010120

Naming convention adjustments.

1.1.0.3:	Boido	010120

Every IO variable is of type BoolIn or BoolOut.
In the future when different types will be needed,
also RealIn,RealOut,IntIn,IntOut etc.. will be added.

1.1.1.4:	Boido	010120

New StepWorkerLib v:1033, naming conventions fixes and IO adjustments

1.1.2.5:	Boido	020120

Version.txt replaced with Version PRG

1.2.2.6:	Boido	040120

Further implementation of the TransferLine StepChains.

1.3.2.7:	Boido	050120

Further implementation of the TransferLine StepChains.

1.4.2.8:	Boido 070120

Implementation of the SM_LineRegulator
*)

END_PROGRAM

// ---- VISUs/Visualization.TcVIS
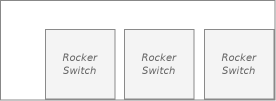
VISUALIZATION Visualization  // 276x101
    RockerSwitch (45,29 70x70), tooltip "'Transfer line 1'", variable: Visu.bStartTL1, behaviour: TOGGLE, style: Switch-RockerSwitch-Blue
    RockerSwitch (124,29 70x70), tooltip "'Transfer line 2'", variable: Visu.bStartTL2, behaviour: TOGGLE, style: Switch-RockerSwitch-Blue
    RockerSwitch (204,29 70x70), tooltip "'Transfer line 3'", variable: Visu.bStartTL3, behaviour: TOGGLE, style: Switch-RockerSwitch-Blue
END_VISUALIZATION
